Staubli VAL3: cycle_putProg.pgx

program cycle_putProg(string x_sName (dimensions=1), num x_nType (dimensions=1))
  local bool l_bFound
begin
  //
  // insert one program at the end of the process List
  // 0 -start list
  // 1 -production list
  // 2 -end list
  //
  if saveData:bDebug
    logMsg("[KERNEL] PLC:Insert program: "+x_sName)
  endIf
  // check before if exist
  call cycle_isFound(x_sName,l_bFound)
  if l_bFound
    call processList:insertCycle(-1,x_sName,1,0,x_nType)
    // check to save or not in order to have the same process next boot
    // call processList:save()
  elseIf saveData:bDebug
    ? "[KERNEL] PLC: "+x_sName+" not found in the program List"
  endIf
end
